% RSLogix 500 project Ladder_Logic.RSS, saved by version 8.30.00.16 %
PROJECT "BBOURBON"    % processor: Bul.1763 MicroLogix 1100 Series B %

PROGRAM FILES
  LAD 2 "MAIN"  12 rungs  % Main Ladder That Calls LAD 3 to 11 Subroutines %
  LAD 3 "RO REQUEST"  8 rungs  % Pounds of RO Water Available for Use %
  LAD 4 "SELECT CIS"  3 rungs  % Select Cistern 1 to 8  to Pump To %
  LAD 5 "FAULTS"  3 rungs  % High Level Faults on Cisterns 1 to 8 %
  LAD 6 "RO VALVES"  10 rungs  % Opens Corresponding Valve After Cistern Is Selecte %
  LAD 7 "RO PUMPING"  10 rungs  % Pounds of RO Water Pumping Based on Flow Sensor %
  LAD 8 "RO TO CIST"  10 rungs  % Monitor RO Water Pumped to Selected Cistern %
  LAD 9 "LOAD CELLS"  26 rungs  % Load Cells for Cisterns 1 to 8 %
  LAD 10 "CALC RO LB"  18 rungs  % Calculate RO Water Pounds, Density Lookup Table %
  LAD 11 "INIT SIMUL"  13 rungs  % Initialize Simulation to Restart From Known Data %

DATA FILES
  O0 OUTPUT  4 elements
  I1 INPUT  6 elements
  S2 STATUS  66 elements
  B3 BINARY  5 elements
  T4 TIMER  2 elements
  C5 COUNTER  1 elements
  R6 CONTROL  1 elements
  N7 INTEGER  11 elements
  F8 FLOAT  120 elements

LADDER 2 "MAIN"    % Main Ladder That Calls LAD 3 to 11 Subroutines %
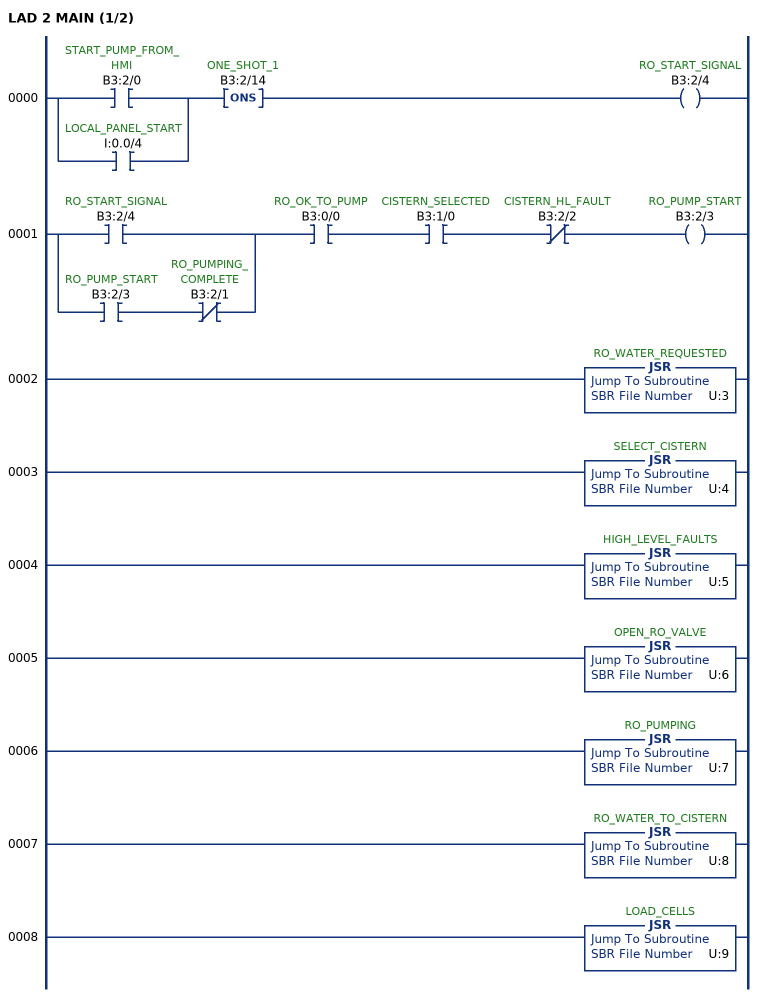
% Rung: 0 %
SOR BST XIC B3:2/0 NXB XIC I:0.0/4 BND ONS B3:2/14 OTE B3:2/4 EOR
%   B3:2/0  START_PUMP_FROM_HMI %
%   I:0.0/4  LOCAL_PANEL_START %
%   B3:2/14  ONE_SHOT_1 %
%   B3:2/4  RO_START_SIGNAL %
% Rung: 1 %
SOR BST XIC B3:2/4 NXB XIC B3:2/3 XIO B3:2/1 BND XIC B3:0/0 XIC B3:1/0 XIO B3:2/2 OTE B3:2/3 EOR
%   B3:2/4  RO_START_SIGNAL %
%   B3:2/3  RO_PUMP_START %
%   B3:2/1  RO_PUMPING_COMPLETE %
%   B3:0/0  RO_OK_TO_PUMP %
%   B3:1/0  CISTERN_SELECTED %
%   B3:2/2  CISTERN_HL_FAULT %
% Rung: 2 %
SOR JSR U:3 EOR
%   U:3  RO_WATER_REQUESTED %
% Rung: 3 %
SOR JSR U:4 EOR
%   U:4  SELECT_CISTERN %
% Rung: 4 %
SOR JSR U:5 EOR
%   U:5  HIGH_LEVEL_FAULTS %
% Rung: 5 %
SOR JSR U:6 EOR
%   U:6  OPEN_RO_VALVE %
% Rung: 6 %
SOR JSR U:7 EOR
%   U:7  RO_PUMPING %
% Rung: 7 %
SOR JSR U:8 EOR
%   U:8  RO_WATER_TO_CISTERN %
% Rung: 8 %
SOR JSR U:9 EOR
%   U:9  LOAD_CELLS %

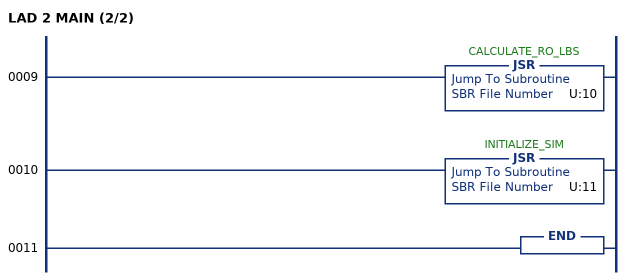
% Rung: 9 %
SOR JSR U:10 EOR
%   U:10  CALCULATE_RO_LBS %
% Rung: 10 %
SOR JSR U:11 EOR
%   U:11  INITIALIZE_SIM %
% Rung: 11 %
SOR END EOR

LADDER 3 "RO REQUEST"    % Pounds of RO Water Available for Use %
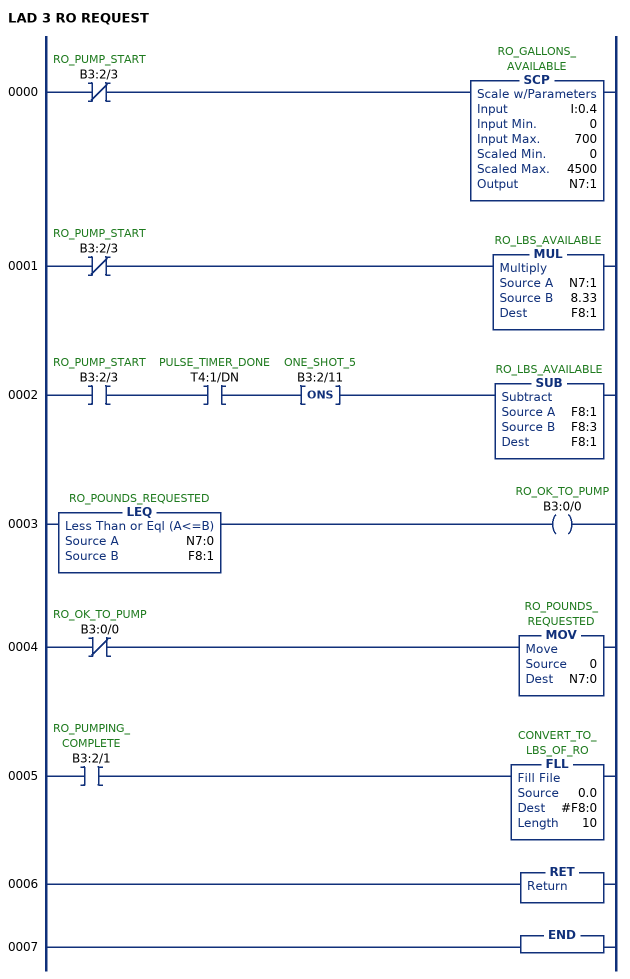
% Rung: 0 %
SOR XIO B3:2/3 SCP I:0.4 0 700 0 4500 N7:1 EOR
%   B3:2/3  RO_PUMP_START %
%   I:0.4  RO_WATER_LEVEL %
%   N7:1  RO_GALLONS_AVAILABLE %
% Rung: 1 %
SOR XIO B3:2/3 MUL N7:1 8.33 F8:1 EOR
%   B3:2/3  RO_PUMP_START %
%   N7:1  RO_GALLONS_AVAILABLE %
%   F8:1  RO_LBS_AVAILABLE %
% Rung: 2 %
SOR XIC B3:2/3 XIC T4:1/DN ONS B3:2/11 SUB F8:1 F8:3 F8:1 EOR
%   B3:2/3  RO_PUMP_START %
%   T4:1/DN  PULSE_TIMER_DONE %
%   B3:2/11  ONE_SHOT_5 %
%   F8:1  RO_LBS_AVAILABLE %
%   F8:3  RO_LBS_PER_TENTH_SEC %
% Rung: 3 %
SOR LEQ N7:0 F8:1 OTE B3:0/0 EOR
%   N7:0  RO_POUNDS_REQUESTED %
%   F8:1  RO_LBS_AVAILABLE %
%   B3:0/0  RO_OK_TO_PUMP %
% Rung: 4 %
SOR XIO B3:0/0 MOV 0 N7:0 EOR
%   B3:0/0  RO_OK_TO_PUMP %
%   N7:0  RO_POUNDS_REQUESTED %
% Rung: 5 %
SOR XIC B3:2/1 FLL 0.0 #F8:0 10 EOR
%   B3:2/1  RO_PUMPING_COMPLETE %
%   F8:0  CONVERT_TO_LBS_OF_RO %
% Rung: 6 %
SOR RET EOR
% Rung: 7 %
SOR END EOR

LADDER 4 "SELECT CIS"    % Select Cistern 1 to 8  to Pump To %
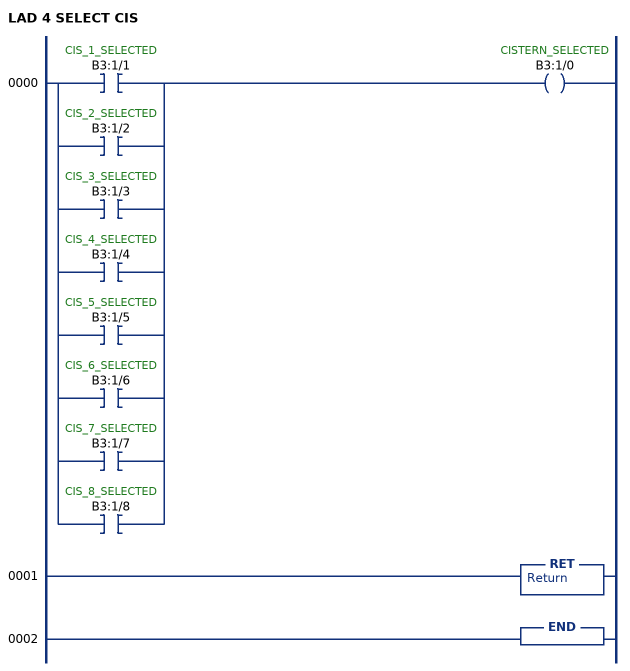
% Rung: 0 %
SOR BST XIC B3:1/1 NXB XIC B3:1/2 NXB XIC B3:1/3 NXB XIC B3:1/4 NXB XIC B3:1/5 NXB XIC B3:1/6 NXB XIC B3:1/7 NXB XIC B3:1/8 BND OTE B3:1/0 EOR
%   B3:1/1  CIS_1_SELECTED %
%   B3:1/2  CIS_2_SELECTED %
%   B3:1/3  CIS_3_SELECTED %
%   B3:1/4  CIS_4_SELECTED %
%   B3:1/5  CIS_5_SELECTED %
%   B3:1/6  CIS_6_SELECTED %
%   B3:1/7  CIS_7_SELECTED %
%   B3:1/8  CIS_8_SELECTED %
%   B3:1/0  CISTERN_SELECTED %
% Rung: 1 %
SOR RET EOR
% Rung: 2 %
SOR END EOR

LADDER 5 "FAULTS"    % High Level Faults on Cisterns 1 to 8 %
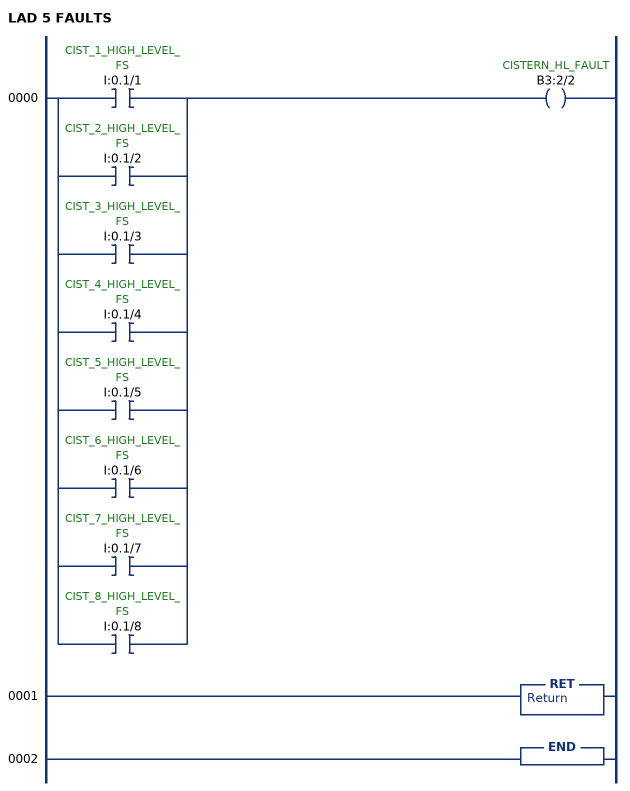
% Rung: 0 %
SOR BST XIC I:0.1/1 NXB XIC I:0.1/2 NXB XIC I:0.1/3 NXB XIC I:0.1/4 NXB XIC I:0.1/5 NXB XIC I:0.1/6 NXB XIC I:0.1/7 NXB XIC I:0.1/8 BND OTE B3:2/2 EOR
%   I:0.1/1  CIST_1_HIGH_LEVEL_FS %
%   I:0.1/2  CIST_2_HIGH_LEVEL_FS %
%   I:0.1/3  CIST_3_HIGH_LEVEL_FS %
%   I:0.1/4  CIST_4_HIGH_LEVEL_FS %
%   I:0.1/5  CIST_5_HIGH_LEVEL_FS %
%   I:0.1/6  CIST_6_HIGH_LEVEL_FS %
%   I:0.1/7  CIST_7_HIGH_LEVEL_FS %
%   I:0.1/8  CIST_8_HIGH_LEVEL_FS %
%   B3:2/2  CISTERN_HL_FAULT %
% Rung: 1 %
SOR RET EOR
% Rung: 2 %
SOR END EOR

LADDER 6 "RO VALVES"    % Opens Corresponding Valve After Cistern Is Selecte %
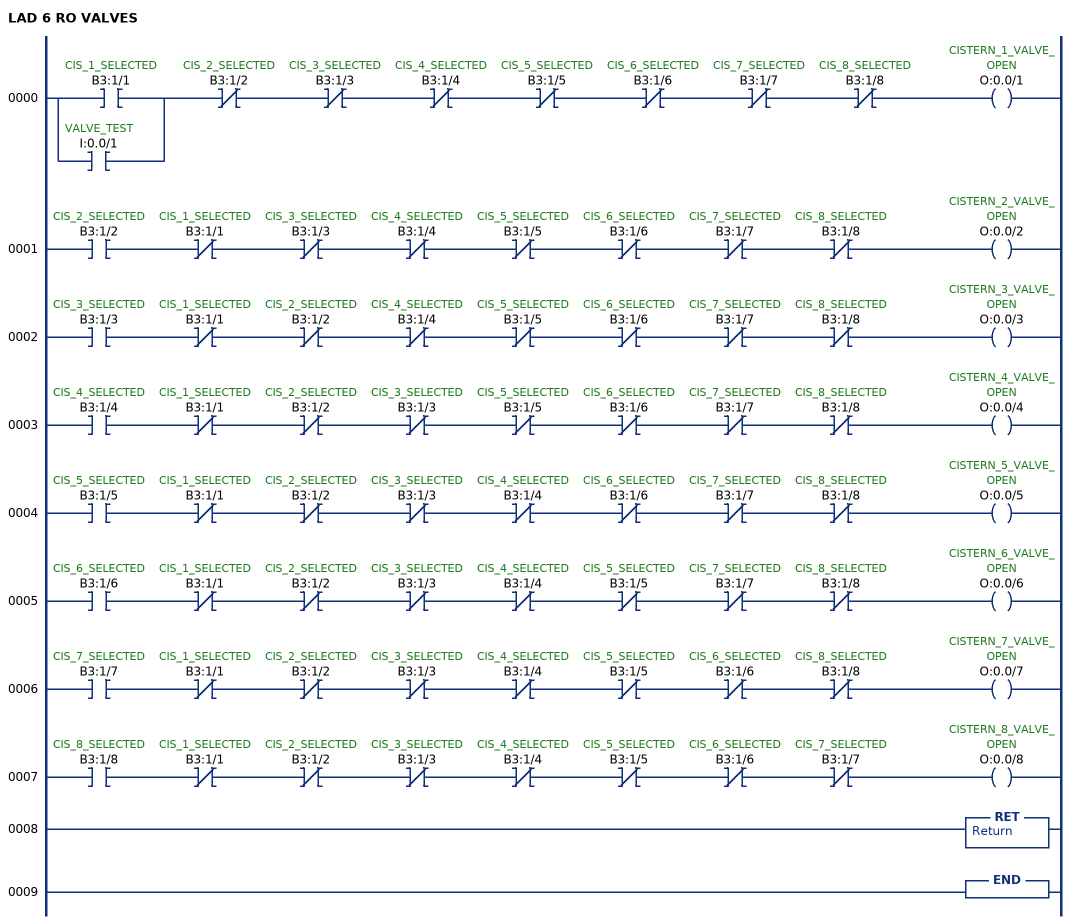
% Rung: 0 %
SOR BST XIC B3:1/1 NXB XIC I:0.0/1 BND XIO B3:1/2 XIO B3:1/3 XIO B3:1/4 XIO B3:1/5 XIO B3:1/6 XIO B3:1/7 XIO B3:1/8 OTE O:0.0/1 EOR
%   B3:1/1  CIS_1_SELECTED %
%   I:0.0/1  VALVE_TEST %
%   B3:1/2  CIS_2_SELECTED %
%   B3:1/3  CIS_3_SELECTED %
%   B3:1/4  CIS_4_SELECTED %
%   B3:1/5  CIS_5_SELECTED %
%   B3:1/6  CIS_6_SELECTED %
%   B3:1/7  CIS_7_SELECTED %
%   B3:1/8  CIS_8_SELECTED %
%   O:0.0/1  CISTERN_1_VALVE_OPEN %
% Rung: 1 %
SOR XIC B3:1/2 XIO B3:1/1 XIO B3:1/3 XIO B3:1/4 XIO B3:1/5 XIO B3:1/6 XIO B3:1/7 XIO B3:1/8 OTE O:0.0/2 EOR
%   B3:1/2  CIS_2_SELECTED %
%   B3:1/1  CIS_1_SELECTED %
%   B3:1/3  CIS_3_SELECTED %
%   B3:1/4  CIS_4_SELECTED %
%   B3:1/5  CIS_5_SELECTED %
%   B3:1/6  CIS_6_SELECTED %
%   B3:1/7  CIS_7_SELECTED %
%   B3:1/8  CIS_8_SELECTED %
%   O:0.0/2  CISTERN_2_VALVE_OPEN %
% Rung: 2 %
SOR XIC B3:1/3 XIO B3:1/1 XIO B3:1/2 XIO B3:1/4 XIO B3:1/5 XIO B3:1/6 XIO B3:1/7 XIO B3:1/8 OTE O:0.0/3 EOR
%   B3:1/3  CIS_3_SELECTED %
%   B3:1/1  CIS_1_SELECTED %
%   B3:1/2  CIS_2_SELECTED %
%   B3:1/4  CIS_4_SELECTED %
%   B3:1/5  CIS_5_SELECTED %
%   B3:1/6  CIS_6_SELECTED %
%   B3:1/7  CIS_7_SELECTED %
%   B3:1/8  CIS_8_SELECTED %
%   O:0.0/3  CISTERN_3_VALVE_OPEN %
% Rung: 3 %
SOR XIC B3:1/4 XIO B3:1/1 XIO B3:1/2 XIO B3:1/3 XIO B3:1/5 XIO B3:1/6 XIO B3:1/7 XIO B3:1/8 OTE O:0.0/4 EOR
%   B3:1/4  CIS_4_SELECTED %
%   B3:1/1  CIS_1_SELECTED %
%   B3:1/2  CIS_2_SELECTED %
%   B3:1/3  CIS_3_SELECTED %
%   B3:1/5  CIS_5_SELECTED %
%   B3:1/6  CIS_6_SELECTED %
%   B3:1/7  CIS_7_SELECTED %
%   B3:1/8  CIS_8_SELECTED %
%   O:0.0/4  CISTERN_4_VALVE_OPEN %
% Rung: 4 %
SOR XIC B3:1/5 XIO B3:1/1 XIO B3:1/2 XIO B3:1/3 XIO B3:1/4 XIO B3:1/6 XIO B3:1/7 XIO B3:1/8 OTE O:0.0/5 EOR
%   B3:1/5  CIS_5_SELECTED %
%   B3:1/1  CIS_1_SELECTED %
%   B3:1/2  CIS_2_SELECTED %
%   B3:1/3  CIS_3_SELECTED %
%   B3:1/4  CIS_4_SELECTED %
%   B3:1/6  CIS_6_SELECTED %
%   B3:1/7  CIS_7_SELECTED %
%   B3:1/8  CIS_8_SELECTED %
%   O:0.0/5  CISTERN_5_VALVE_OPEN %
% Rung: 5 %
SOR XIC B3:1/6 XIO B3:1/1 XIO B3:1/2 XIO B3:1/3 XIO B3:1/4 XIO B3:1/5 XIO B3:1/7 XIO B3:1/8 OTE O:0.0/6 EOR
%   B3:1/6  CIS_6_SELECTED %
%   B3:1/1  CIS_1_SELECTED %
%   B3:1/2  CIS_2_SELECTED %
%   B3:1/3  CIS_3_SELECTED %
%   B3:1/4  CIS_4_SELECTED %
%   B3:1/5  CIS_5_SELECTED %
%   B3:1/7  CIS_7_SELECTED %
%   B3:1/8  CIS_8_SELECTED %
%   O:0.0/6  CISTERN_6_VALVE_OPEN %
% Rung: 6 %
SOR XIC B3:1/7 XIO B3:1/1 XIO B3:1/2 XIO B3:1/3 XIO B3:1/4 XIO B3:1/5 XIO B3:1/6 XIO B3:1/8 OTE O:0.0/7 EOR
%   B3:1/7  CIS_7_SELECTED %
%   B3:1/1  CIS_1_SELECTED %
%   B3:1/2  CIS_2_SELECTED %
%   B3:1/3  CIS_3_SELECTED %
%   B3:1/4  CIS_4_SELECTED %
%   B3:1/5  CIS_5_SELECTED %
%   B3:1/6  CIS_6_SELECTED %
%   B3:1/8  CIS_8_SELECTED %
%   O:0.0/7  CISTERN_7_VALVE_OPEN %
% Rung: 7 %
SOR XIC B3:1/8 XIO B3:1/1 XIO B3:1/2 XIO B3:1/3 XIO B3:1/4 XIO B3:1/5 XIO B3:1/6 XIO B3:1/7 OTE O:0.0/8 EOR
%   B3:1/8  CIS_8_SELECTED %
%   B3:1/1  CIS_1_SELECTED %
%   B3:1/2  CIS_2_SELECTED %
%   B3:1/3  CIS_3_SELECTED %
%   B3:1/4  CIS_4_SELECTED %
%   B3:1/5  CIS_5_SELECTED %
%   B3:1/6  CIS_6_SELECTED %
%   B3:1/7  CIS_7_SELECTED %
%   O:0.0/8  CISTERN_8_VALVE_OPEN %
% Rung: 8 %
SOR RET EOR
% Rung: 9 %
SOR END EOR

LADDER 7 "RO PUMPING"    % Pounds of RO Water Pumping Based on Flow Sensor %
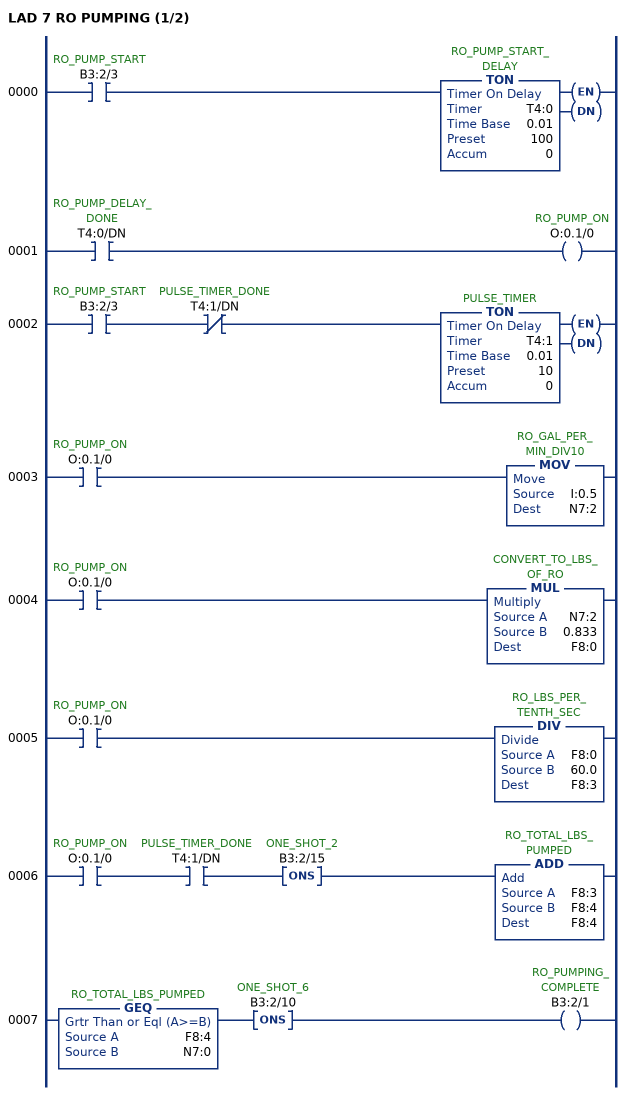
% Rung: 0 %
SOR XIC B3:2/3 TON T4:0 0.01 100 0 EOR
%   B3:2/3  RO_PUMP_START %
%   T4:0  RO_PUMP_START_DELAY %
% Rung: 1 %
SOR XIC T4:0/DN OTE O:0.1/0 EOR
%   T4:0/DN  RO_PUMP_DELAY_DONE %
%   O:0.1/0  RO_PUMP_ON %
% Rung: 2 %
SOR XIC B3:2/3 XIO T4:1/DN TON T4:1 0.01 10 0 EOR
%   B3:2/3  RO_PUMP_START %
%   T4:1/DN  PULSE_TIMER_DONE %
%   T4:1  PULSE_TIMER %
% Rung: 3 %
SOR XIC O:0.1/0 MOV I:0.5 N7:2 EOR
%   O:0.1/0  RO_PUMP_ON %
%   I:0.5  RO_FLOW_SENSOR %
%   N7:2  RO_GAL_PER_MIN_DIV10 %
% Rung: 4 %
SOR XIC O:0.1/0 MUL N7:2 0.833 F8:0 EOR
%   O:0.1/0  RO_PUMP_ON %
%   N7:2  RO_GAL_PER_MIN_DIV10 %
%   F8:0  CONVERT_TO_LBS_OF_RO %
% Rung: 5 %
SOR XIC O:0.1/0 DIV F8:0 60.0 F8:3 EOR
%   O:0.1/0  RO_PUMP_ON %
%   F8:0  CONVERT_TO_LBS_OF_RO %
%   F8:3  RO_LBS_PER_TENTH_SEC %
% Rung: 6 %
SOR XIC O:0.1/0 XIC T4:1/DN ONS B3:2/15 ADD F8:3 F8:4 F8:4 EOR
%   O:0.1/0  RO_PUMP_ON %
%   T4:1/DN  PULSE_TIMER_DONE %
%   B3:2/15  ONE_SHOT_2 %
%   F8:3  RO_LBS_PER_TENTH_SEC %
%   F8:4  RO_TOTAL_LBS_PUMPED %
% Rung: 7 %
SOR GEQ F8:4 N7:0 ONS B3:2/10 OTE B3:2/1 EOR
%   F8:4  RO_TOTAL_LBS_PUMPED %
%   N7:0  RO_POUNDS_REQUESTED %
%   B3:2/10  ONE_SHOT_6 %
%   B3:2/1  RO_PUMPING_COMPLETE %

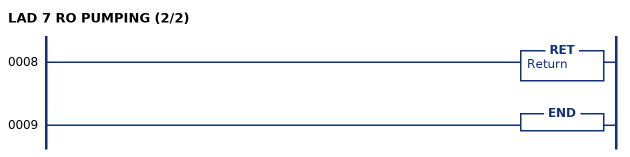
% Rung: 8 %
SOR RET EOR
% Rung: 9 %
SOR END EOR

LADDER 8 "RO TO CIST"    % Monitor RO Water Pumped to Selected Cistern %
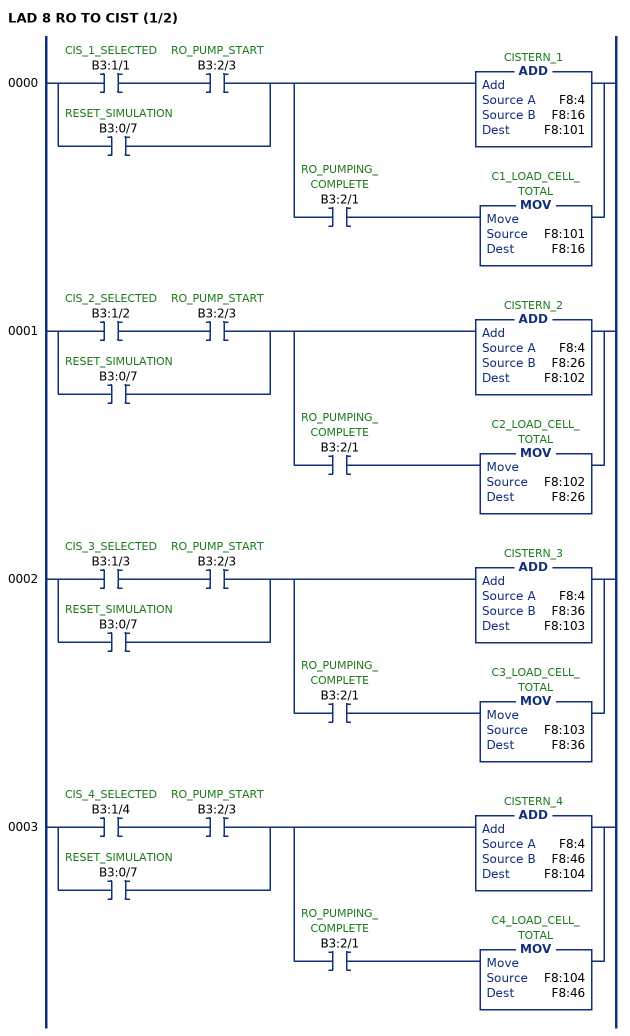
% Rung: 0 %
SOR BST XIC B3:1/1 XIC B3:2/3 NXB XIC B3:0/7 BND BST ADD F8:4 F8:16 F8:101 NXB XIC B3:2/1 MOV F8:101 F8:16 BND EOR
%   B3:1/1  CIS_1_SELECTED %
%   B3:2/3  RO_PUMP_START %
%   B3:0/7  RESET_SIMULATION %
%   F8:4  RO_TOTAL_LBS_PUMPED %
%   F8:16  C1_LOAD_CELL_TOTAL %
%   F8:101  CISTERN_1 %
%   B3:2/1  RO_PUMPING_COMPLETE %
% Rung: 1 %
SOR BST XIC B3:1/2 XIC B3:2/3 NXB XIC B3:0/7 BND BST ADD F8:4 F8:26 F8:102 NXB XIC B3:2/1 MOV F8:102 F8:26 BND EOR
%   B3:1/2  CIS_2_SELECTED %
%   B3:2/3  RO_PUMP_START %
%   B3:0/7  RESET_SIMULATION %
%   F8:4  RO_TOTAL_LBS_PUMPED %
%   F8:26  C2_LOAD_CELL_TOTAL %
%   F8:102  CISTERN_2 %
%   B3:2/1  RO_PUMPING_COMPLETE %
% Rung: 2 %
SOR BST XIC B3:1/3 XIC B3:2/3 NXB XIC B3:0/7 BND BST ADD F8:4 F8:36 F8:103 NXB XIC B3:2/1 MOV F8:103 F8:36 BND EOR
%   B3:1/3  CIS_3_SELECTED %
%   B3:2/3  RO_PUMP_START %
%   B3:0/7  RESET_SIMULATION %
%   F8:4  RO_TOTAL_LBS_PUMPED %
%   F8:36  C3_LOAD_CELL_TOTAL %
%   F8:103  CISTERN_3 %
%   B3:2/1  RO_PUMPING_COMPLETE %
% Rung: 3 %
SOR BST XIC B3:1/4 XIC B3:2/3 NXB XIC B3:0/7 BND BST ADD F8:4 F8:46 F8:104 NXB XIC B3:2/1 MOV F8:104 F8:46 BND EOR
%   B3:1/4  CIS_4_SELECTED %
%   B3:2/3  RO_PUMP_START %
%   B3:0/7  RESET_SIMULATION %
%   F8:4  RO_TOTAL_LBS_PUMPED %
%   F8:46  C4_LOAD_CELL_TOTAL %
%   F8:104  CISTERN_4 %
%   B3:2/1  RO_PUMPING_COMPLETE %

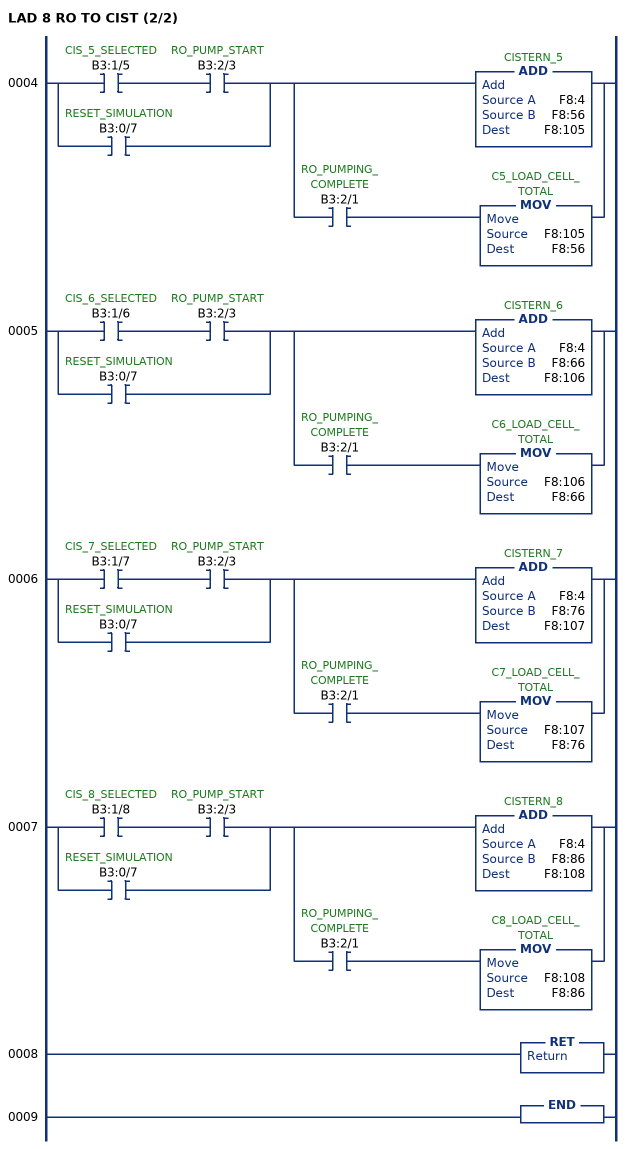
% Rung: 4 %
SOR BST XIC B3:1/5 XIC B3:2/3 NXB XIC B3:0/7 BND BST ADD F8:4 F8:56 F8:105 NXB XIC B3:2/1 MOV F8:105 F8:56 BND EOR
%   B3:1/5  CIS_5_SELECTED %
%   B3:2/3  RO_PUMP_START %
%   B3:0/7  RESET_SIMULATION %
%   F8:4  RO_TOTAL_LBS_PUMPED %
%   F8:56  C5_LOAD_CELL_TOTAL %
%   F8:105  CISTERN_5 %
%   B3:2/1  RO_PUMPING_COMPLETE %
% Rung: 5 %
SOR BST XIC B3:1/6 XIC B3:2/3 NXB XIC B3:0/7 BND BST ADD F8:4 F8:66 F8:106 NXB XIC B3:2/1 MOV F8:106 F8:66 BND EOR
%   B3:1/6  CIS_6_SELECTED %
%   B3:2/3  RO_PUMP_START %
%   B3:0/7  RESET_SIMULATION %
%   F8:4  RO_TOTAL_LBS_PUMPED %
%   F8:66  C6_LOAD_CELL_TOTAL %
%   F8:106  CISTERN_6 %
%   B3:2/1  RO_PUMPING_COMPLETE %
% Rung: 6 %
SOR BST XIC B3:1/7 XIC B3:2/3 NXB XIC B3:0/7 BND BST ADD F8:4 F8:76 F8:107 NXB XIC B3:2/1 MOV F8:107 F8:76 BND EOR
%   B3:1/7  CIS_7_SELECTED %
%   B3:2/3  RO_PUMP_START %
%   B3:0/7  RESET_SIMULATION %
%   F8:4  RO_TOTAL_LBS_PUMPED %
%   F8:76  C7_LOAD_CELL_TOTAL %
%   F8:107  CISTERN_7 %
%   B3:2/1  RO_PUMPING_COMPLETE %
% Rung: 7 %
SOR BST XIC B3:1/8 XIC B3:2/3 NXB XIC B3:0/7 BND BST ADD F8:4 F8:86 F8:108 NXB XIC B3:2/1 MOV F8:108 F8:86 BND EOR
%   B3:1/8  CIS_8_SELECTED %
%   B3:2/3  RO_PUMP_START %
%   B3:0/7  RESET_SIMULATION %
%   F8:4  RO_TOTAL_LBS_PUMPED %
%   F8:86  C8_LOAD_CELL_TOTAL %
%   F8:108  CISTERN_8 %
%   B3:2/1  RO_PUMPING_COMPLETE %
% Rung: 8 %
SOR RET EOR
% Rung: 9 %
SOR END EOR

LADDER 9 "LOAD CELLS"    % Load Cells for Cisterns 1 to 8 %
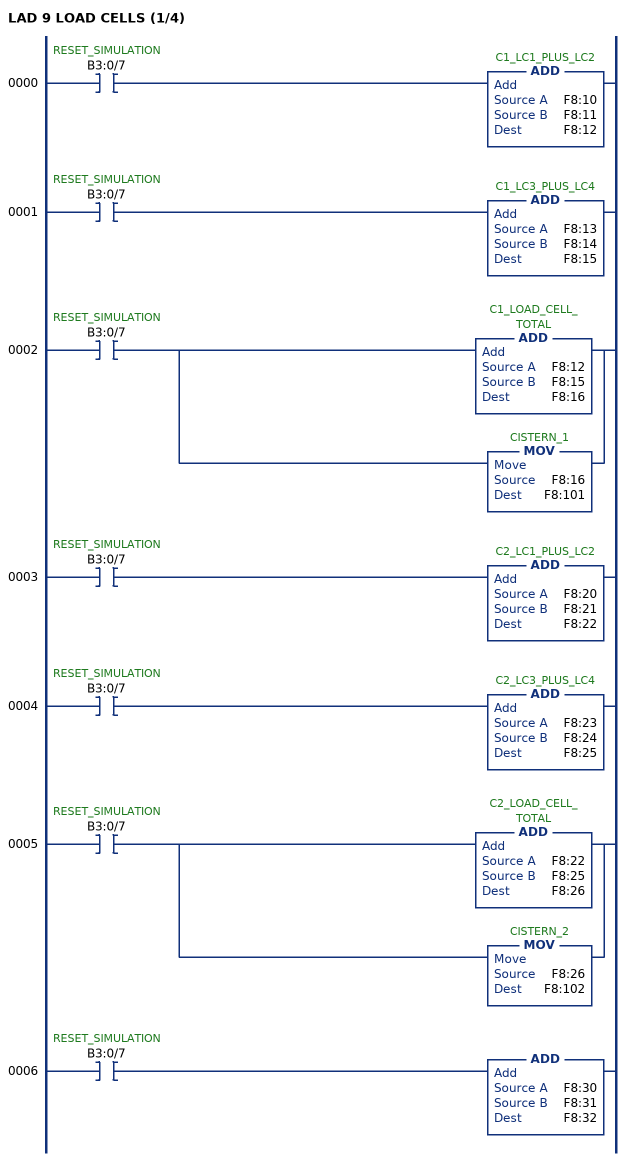
% Rung: 0 %
SOR XIC B3:0/7 ADD F8:10 F8:11 F8:12 EOR
%   B3:0/7  RESET_SIMULATION %
%   F8:10  C1_LOAD_CELL_1 %
%   F8:11  C1_LOAD_CELL_2 %
%   F8:12  C1_LC1_PLUS_LC2 %
% Rung: 1 %
SOR XIC B3:0/7 ADD F8:13 F8:14 F8:15 EOR
%   B3:0/7  RESET_SIMULATION %
%   F8:13  C1_LOAD_CELL_3 %
%   F8:14  C1_LOAD_CELL_4 %
%   F8:15  C1_LC3_PLUS_LC4 %
% Rung: 2 %
SOR XIC B3:0/7 BST ADD F8:12 F8:15 F8:16 NXB MOV F8:16 F8:101 BND EOR
%   B3:0/7  RESET_SIMULATION %
%   F8:12  C1_LC1_PLUS_LC2 %
%   F8:15  C1_LC3_PLUS_LC4 %
%   F8:16  C1_LOAD_CELL_TOTAL %
%   F8:101  CISTERN_1 %
% Rung: 3 %
SOR XIC B3:0/7 ADD F8:20 F8:21 F8:22 EOR
%   B3:0/7  RESET_SIMULATION %
%   F8:20  C2_LOAD_CELL_1 %
%   F8:21  C2_LOAD_CELL_2 %
%   F8:22  C2_LC1_PLUS_LC2 %
% Rung: 4 %
SOR XIC B3:0/7 ADD F8:23 F8:24 F8:25 EOR
%   B3:0/7  RESET_SIMULATION %
%   F8:23  C2_LOAD_CELL_3 %
%   F8:24  C2_LOAD_CELL_4 %
%   F8:25  C2_LC3_PLUS_LC4 %
% Rung: 5 %
SOR XIC B3:0/7 BST ADD F8:22 F8:25 F8:26 NXB MOV F8:26 F8:102 BND EOR
%   B3:0/7  RESET_SIMULATION %
%   F8:22  C2_LC1_PLUS_LC2 %
%   F8:25  C2_LC3_PLUS_LC4 %
%   F8:26  C2_LOAD_CELL_TOTAL %
%   F8:102  CISTERN_2 %
% Rung: 6 %
SOR XIC B3:0/7 ADD F8:30 F8:31 F8:32 EOR
%   B3:0/7  RESET_SIMULATION %
%   F8:30  C3_LOAD_CELL_1 %

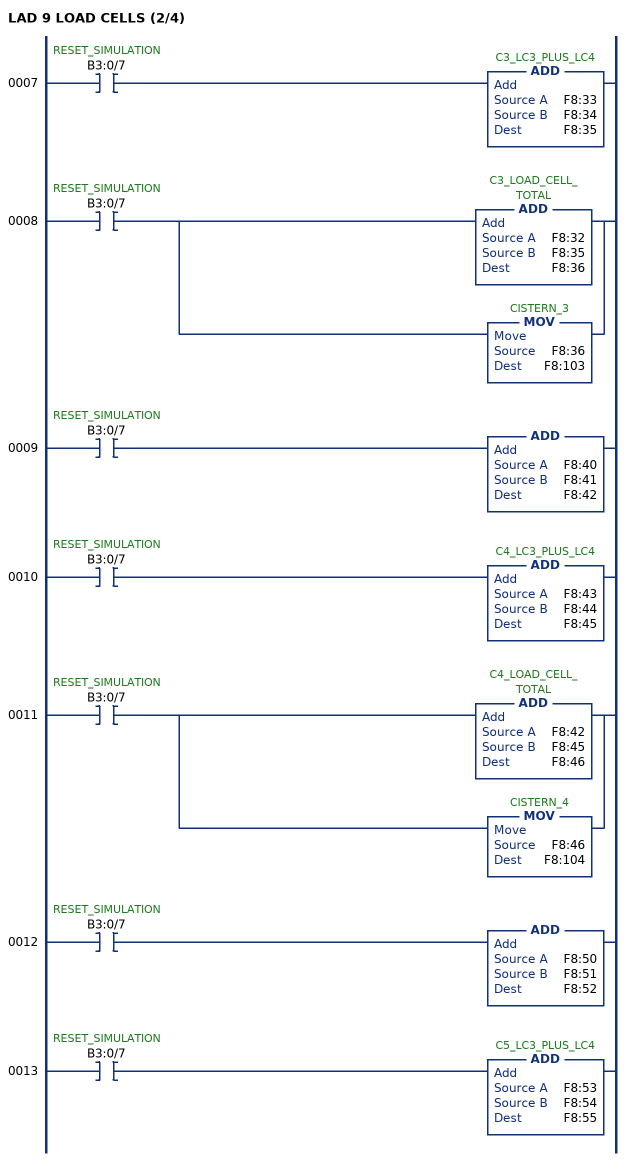
% Rung: 7 %
SOR XIC B3:0/7 ADD F8:33 F8:34 F8:35 EOR
%   B3:0/7  RESET_SIMULATION %
%   F8:35  C3_LC3_PLUS_LC4 %
% Rung: 8 %
SOR XIC B3:0/7 BST ADD F8:32 F8:35 F8:36 NXB MOV F8:36 F8:103 BND EOR
%   B3:0/7  RESET_SIMULATION %
%   F8:35  C3_LC3_PLUS_LC4 %
%   F8:36  C3_LOAD_CELL_TOTAL %
%   F8:103  CISTERN_3 %
% Rung: 9 %
SOR XIC B3:0/7 ADD F8:40 F8:41 F8:42 EOR
%   B3:0/7  RESET_SIMULATION %
%   F8:40  C4_LOAD_CELL_1 %
% Rung: 10 %
SOR XIC B3:0/7 ADD F8:43 F8:44 F8:45 EOR
%   B3:0/7  RESET_SIMULATION %
%   F8:45  C4_LC3_PLUS_LC4 %
% Rung: 11 %
SOR XIC B3:0/7 BST ADD F8:42 F8:45 F8:46 NXB MOV F8:46 F8:104 BND EOR
%   B3:0/7  RESET_SIMULATION %
%   F8:45  C4_LC3_PLUS_LC4 %
%   F8:46  C4_LOAD_CELL_TOTAL %
%   F8:104  CISTERN_4 %
% Rung: 12 %
SOR XIC B3:0/7 ADD F8:50 F8:51 F8:52 EOR
%   B3:0/7  RESET_SIMULATION %
%   F8:50  C5_LOAD_CELL_1 %
% Rung: 13 %
SOR XIC B3:0/7 ADD F8:53 F8:54 F8:55 EOR
%   B3:0/7  RESET_SIMULATION %
%   F8:55  C5_LC3_PLUS_LC4 %

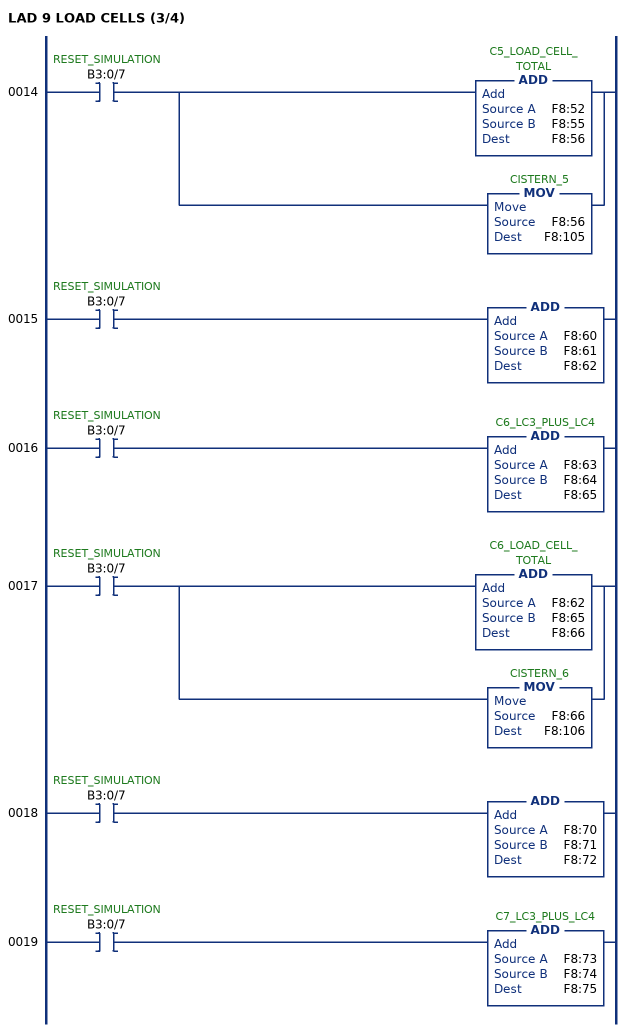
% Rung: 14 %
SOR XIC B3:0/7 BST ADD F8:52 F8:55 F8:56 NXB MOV F8:56 F8:105 BND EOR
%   B3:0/7  RESET_SIMULATION %
%   F8:55  C5_LC3_PLUS_LC4 %
%   F8:56  C5_LOAD_CELL_TOTAL %
%   F8:105  CISTERN_5 %
% Rung: 15 %
SOR XIC B3:0/7 ADD F8:60 F8:61 F8:62 EOR
%   B3:0/7  RESET_SIMULATION %
%   F8:60  C6_LOAD_CELL_1 %
% Rung: 16 %
SOR XIC B3:0/7 ADD F8:63 F8:64 F8:65 EOR
%   B3:0/7  RESET_SIMULATION %
%   F8:65  C6_LC3_PLUS_LC4 %
% Rung: 17 %
SOR XIC B3:0/7 BST ADD F8:62 F8:65 F8:66 NXB MOV F8:66 F8:106 BND EOR
%   B3:0/7  RESET_SIMULATION %
%   F8:65  C6_LC3_PLUS_LC4 %
%   F8:66  C6_LOAD_CELL_TOTAL %
%   F8:106  CISTERN_6 %
% Rung: 18 %
SOR XIC B3:0/7 ADD F8:70 F8:71 F8:72 EOR
%   B3:0/7  RESET_SIMULATION %
%   F8:70  C7_LOAD_CELL_1 %
% Rung: 19 %
SOR XIC B3:0/7 ADD F8:73 F8:74 F8:75 EOR
%   B3:0/7  RESET_SIMULATION %
%   F8:75  C7_LC3_PLUS_LC4 %

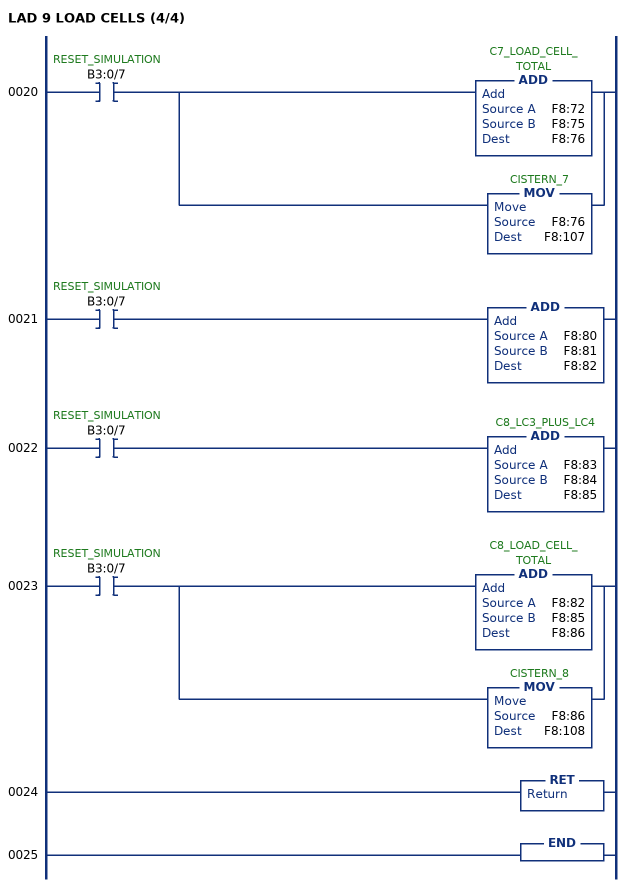
% Rung: 20 %
SOR XIC B3:0/7 BST ADD F8:72 F8:75 F8:76 NXB MOV F8:76 F8:107 BND EOR
%   B3:0/7  RESET_SIMULATION %
%   F8:75  C7_LC3_PLUS_LC4 %
%   F8:76  C7_LOAD_CELL_TOTAL %
%   F8:107  CISTERN_7 %
% Rung: 21 %
SOR XIC B3:0/7 ADD F8:80 F8:81 F8:82 EOR
%   B3:0/7  RESET_SIMULATION %
%   F8:80  C8_LOAD_CELL_1 %
% Rung: 22 %
SOR XIC B3:0/7 ADD F8:83 F8:84 F8:85 EOR
%   B3:0/7  RESET_SIMULATION %
%   F8:85  C8_LC3_PLUS_LC4 %
% Rung: 23 %
SOR XIC B3:0/7 BST ADD F8:82 F8:85 F8:86 NXB MOV F8:86 F8:108 BND EOR
%   B3:0/7  RESET_SIMULATION %
%   F8:85  C8_LC3_PLUS_LC4 %
%   F8:86  C8_LOAD_CELL_TOTAL %
%   F8:108  CISTERN_8 %
% Rung: 24 %
SOR RET EOR
% Rung: 25 %
SOR END EOR

LADDER 10 "CALC RO LB"    % Calculate RO Water Pounds, Density Lookup Table %
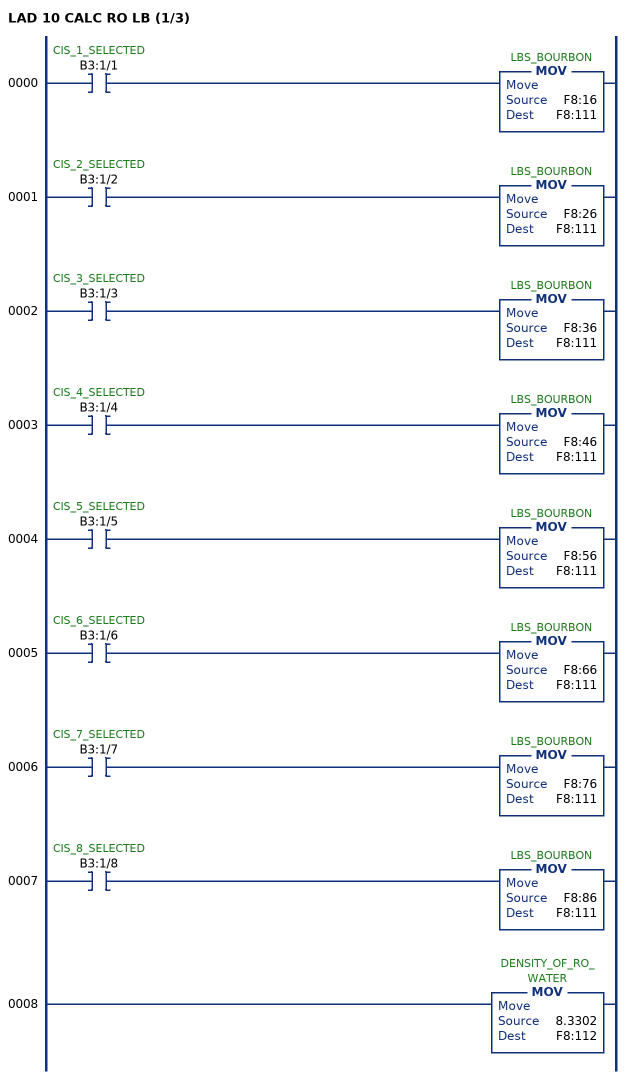
% Rung: 0 %
SOR XIC B3:1/1 MOV F8:16 F8:111 EOR
%   B3:1/1  CIS_1_SELECTED %
%   F8:16  C1_LOAD_CELL_TOTAL %
%   F8:111  LBS_BOURBON %
% Rung: 1 %
SOR XIC B3:1/2 MOV F8:26 F8:111 EOR
%   B3:1/2  CIS_2_SELECTED %
%   F8:26  C2_LOAD_CELL_TOTAL %
%   F8:111  LBS_BOURBON %
% Rung: 2 %
SOR XIC B3:1/3 MOV F8:36 F8:111 EOR
%   B3:1/3  CIS_3_SELECTED %
%   F8:36  C3_LOAD_CELL_TOTAL %
%   F8:111  LBS_BOURBON %
% Rung: 3 %
SOR XIC B3:1/4 MOV F8:46 F8:111 EOR
%   B3:1/4  CIS_4_SELECTED %
%   F8:46  C4_LOAD_CELL_TOTAL %
%   F8:111  LBS_BOURBON %
% Rung: 4 %
SOR XIC B3:1/5 MOV F8:56 F8:111 EOR
%   B3:1/5  CIS_5_SELECTED %
%   F8:56  C5_LOAD_CELL_TOTAL %
%   F8:111  LBS_BOURBON %
% Rung: 5 %
SOR XIC B3:1/6 MOV F8:66 F8:111 EOR
%   B3:1/6  CIS_6_SELECTED %
%   F8:66  C6_LOAD_CELL_TOTAL %
%   F8:111  LBS_BOURBON %
% Rung: 6 %
SOR XIC B3:1/7 MOV F8:76 F8:111 EOR
%   B3:1/7  CIS_7_SELECTED %
%   F8:76  C7_LOAD_CELL_TOTAL %
%   F8:111  LBS_BOURBON %
% Rung: 7 %
SOR XIC B3:1/8 MOV F8:86 F8:111 EOR
%   B3:1/8  CIS_8_SELECTED %
%   F8:86  C8_LOAD_CELL_TOTAL %
%   F8:111  LBS_BOURBON %
% Rung: 8 %
SOR MOV 8.3302 F8:112 EOR
%   F8:112  DENSITY_OF_RO_WATER %

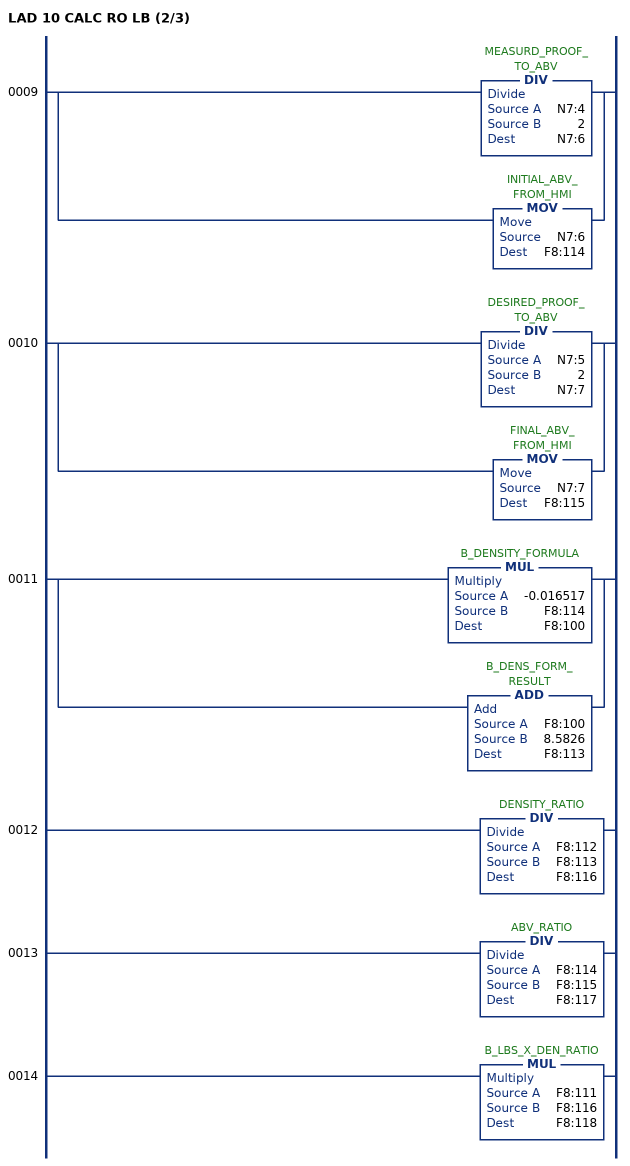
% Rung: 9 %
SOR BST DIV N7:4 2 N7:6 NXB MOV N7:6 F8:114 BND EOR
%   N7:4  INITIAL_MEASURED_ABV %
%   N7:6  MEASURD_PROOF_TO_ABV %
%   F8:114  INITIAL_ABV_FROM_HMI %
% Rung: 10 %
SOR BST DIV N7:5 2 N7:7 NXB MOV N7:7 F8:115 BND EOR
%   N7:5  FINAL_DESIRED_ABV %
%   N7:7  DESIRED_PROOF_TO_ABV %
%   F8:115  FINAL_ABV_FROM_HMI %
% Rung: 11 %
SOR BST MUL -0.016517 F8:114 F8:100 NXB ADD F8:100 8.5826 F8:113 BND EOR
%   F8:114  INITIAL_ABV_FROM_HMI %
%   F8:100  B_DENSITY_FORMULA %
%   F8:113  B_DENS_FORM_RESULT %
% Rung: 12 %
SOR DIV F8:112 F8:113 F8:116 EOR
%   F8:112  DENSITY_OF_RO_WATER %
%   F8:113  B_DENS_FORM_RESULT %
%   F8:116  DENSITY_RATIO %
% Rung: 13 %
SOR DIV F8:114 F8:115 F8:117 EOR
%   F8:114  INITIAL_ABV_FROM_HMI %
%   F8:115  FINAL_ABV_FROM_HMI %
%   F8:117  ABV_RATIO %
% Rung: 14 %
SOR MUL F8:111 F8:116 F8:118 EOR
%   F8:111  LBS_BOURBON %
%   F8:116  DENSITY_RATIO %
%   F8:118  B_LBS_X_DEN_RATIO %

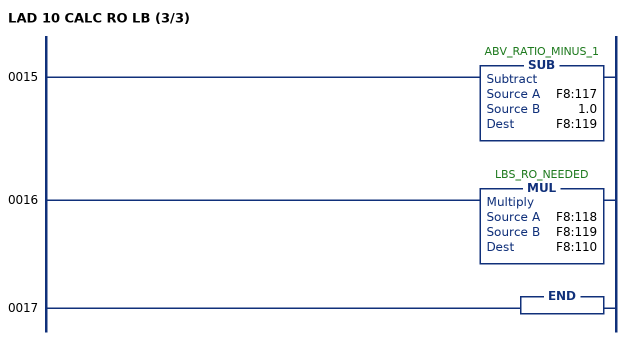
% Rung: 15 %
SOR SUB F8:117 1.0 F8:119 EOR
%   F8:117  ABV_RATIO %
%   F8:119  ABV_RATIO_MINUS_1 %
% Rung: 16 %
SOR MUL F8:118 F8:119 F8:110 EOR
%   F8:118  B_LBS_X_DEN_RATIO %
%   F8:119  ABV_RATIO_MINUS_1 %
%   F8:110  LBS_RO_NEEDED %
% Rung: 17 %
SOR END EOR

LADDER 11 "INIT SIMUL"    % Initialize Simulation to Restart From Known Data %
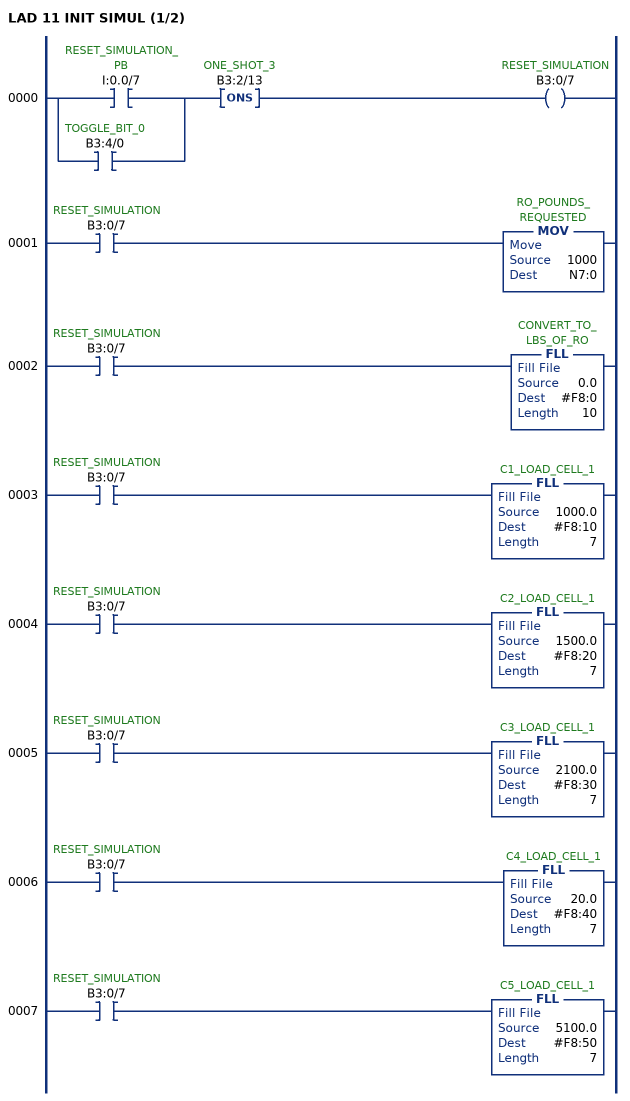
% Rung: 0 %
SOR BST XIC I:0.0/7 NXB XIC B3:4/0 BND ONS B3:2/13 OTE B3:0/7 EOR
%   I:0.0/7  RESET_SIMULATION_PB %
%   B3:4/0  TOGGLE_BIT_0 %
%   B3:2/13  ONE_SHOT_3 %
%   B3:0/7  RESET_SIMULATION %
% Rung: 1 %
SOR XIC B3:0/7 MOV 1000 N7:0 EOR
%   B3:0/7  RESET_SIMULATION %
%   N7:0  RO_POUNDS_REQUESTED %
% Rung: 2 %
SOR XIC B3:0/7 FLL 0.0 #F8:0 10 EOR
%   B3:0/7  RESET_SIMULATION %
%   F8:0  CONVERT_TO_LBS_OF_RO %
% Rung: 3 %
SOR XIC B3:0/7 FLL 1000.0 #F8:10 7 EOR
%   B3:0/7  RESET_SIMULATION %
%   F8:10  C1_LOAD_CELL_1 %
% Rung: 4 %
SOR XIC B3:0/7 FLL 1500.0 #F8:20 7 EOR
%   B3:0/7  RESET_SIMULATION %
%   F8:20  C2_LOAD_CELL_1 %
% Rung: 5 %
SOR XIC B3:0/7 FLL 2100.0 #F8:30 7 EOR
%   B3:0/7  RESET_SIMULATION %
%   F8:30  C3_LOAD_CELL_1 %
% Rung: 6 %
SOR XIC B3:0/7 FLL 20.0 #F8:40 7 EOR
%   B3:0/7  RESET_SIMULATION %
%   F8:40  C4_LOAD_CELL_1 %
% Rung: 7 %
SOR XIC B3:0/7 FLL 5100.0 #F8:50 7 EOR
%   B3:0/7  RESET_SIMULATION %
%   F8:50  C5_LOAD_CELL_1 %

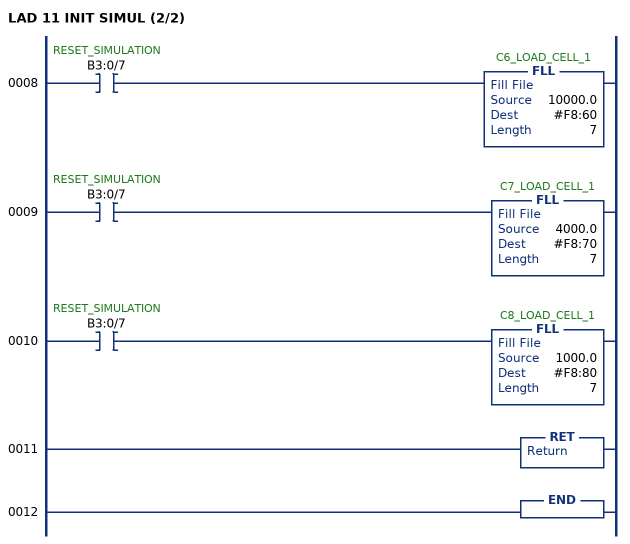
% Rung: 8 %
SOR XIC B3:0/7 FLL 10000.0 #F8:60 7 EOR
%   B3:0/7  RESET_SIMULATION %
%   F8:60  C6_LOAD_CELL_1 %
% Rung: 9 %
SOR XIC B3:0/7 FLL 4000.0 #F8:70 7 EOR
%   B3:0/7  RESET_SIMULATION %
%   F8:70  C7_LOAD_CELL_1 %
% Rung: 10 %
SOR XIC B3:0/7 FLL 1000.0 #F8:80 7 EOR
%   B3:0/7  RESET_SIMULATION %
%   F8:80  C8_LOAD_CELL_1 %
% Rung: 11 %
SOR RET EOR
% Rung: 12 %
SOR END EOR

OTHER DOCUMENTED ADDRESSES
  B3:2/12  ONE_SHOT_4
  F9:[N7:4]  LOOK_UP_DENSITY
  PFILE:4  "Select Cistern to Pu mp Into"
  PFILE:6  "After Cistern is Sel ected Open Correspon ding Valve"
  PFILE:7  "Pounds of RO Water P umped Based on Flow Sensor"
  PFILE:8  "Monitor RO Water to Selected Cistern"
  PFILE:10  "Reset Simulation"

DATA TABLE (non-zero values as saved)
DATA B3
% B3:0 % 0X8401 0X0003 0X0000 0X0000 0X0000
DATA T4
% .PRE .ACC %
% T4:0 % 100 0
% T4:1 % 10 0
DATA C5
% .PRE .ACC %
% C5:0 % 32767 1892
DATA N7
% N7:0 % 1000 4686 635 0 120 80 60 40 0 0
DATA F8
% F8:0 % 0 39034.38 0 0 0
% F8:10 % 1000 1000 2000 1000 1000
% F8:15 % 2000 4000 0 0 0
% F8:20 % 1500 1500 3000 1500 1500
% F8:25 % 3000 6000 0 0 0
% F8:30 % 2100 2100 4200 2100 2100
% F8:35 % 4200 8400 0 0 0
% F8:40 % 20 20 40 20 20
% F8:45 % 40 80 0 0 0
% F8:50 % 5100 5100 10200 5100 5100
% F8:55 % 10200 20400 0 0 0
% F8:60 % 10000 10000 20000 10000 10000
% F8:65 % 20000 40000 0 0 0
% F8:70 % 4000 4000 8000 4000 4000
% F8:75 % 8000 16000 0 0 0
% F8:80 % 1000 1000 2000 1000 1000
% F8:85 % 2000 4000 0 0 0
% F8:100 % -0.99102 4000 6000 8400 80
% F8:105 % 20400 40000 16000 4000 0
% F8:110 % 2194.589 4000 8.3302 7.591579 60
% F8:115 % 40 1.097295 1.5 4389.179 0.5
